// Mitsubishi GX Works2 project: infinite   PLC: Q03UDV

PROGRAM MAIN
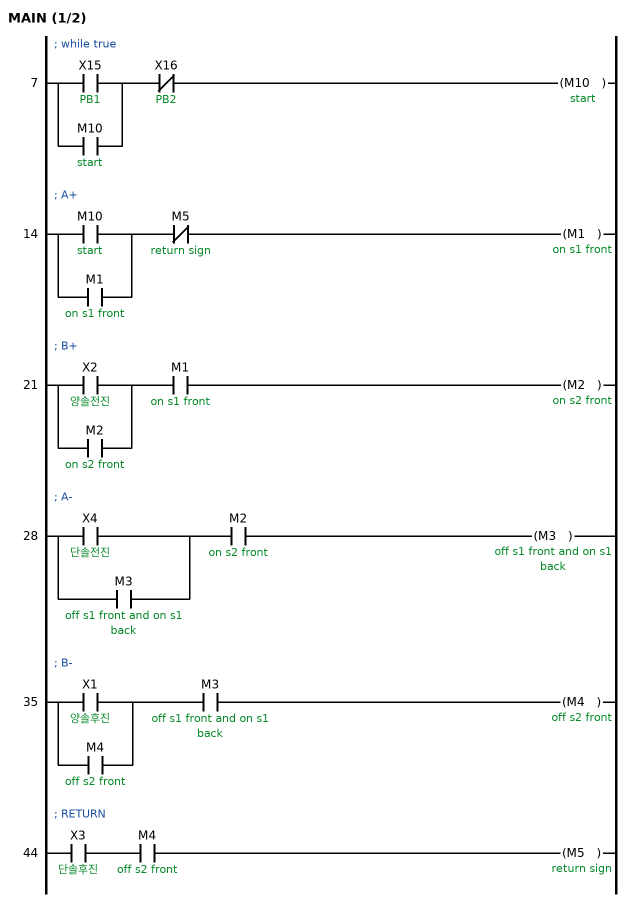
; while true
7     LD      X15  ; PB1
      OR      M10  ; start
      ANI     X16  ; PB2
      OUT     M10  ; start
; A+
14    LD      M10  ; start
      OR      M1  ; on s1 front
      ANI     M5  ; return sign
      OUT     M1  ; on s1 front
; B+
21    LD      X2  ; 양솔전진
      OR      M2  ; on s2 front
      AND     M1  ; on s1 front
      OUT     M2  ; on s2 front
; A-
28    LD      X4  ; 단솔전진
      OR      M3  ; off s1 front and on s1 back
      AND     M2  ; on s2 front
      OUT     M3  ; off s1 front and on s1 back
; B-
35    LD      X1  ; 양솔후진
      OR      M4  ; off s2 front
      AND     M3  ; off s1 front and on s1 back
      OUT     M4  ; off s2 front
; RETURN
44    LD      X3  ; 단솔후진
      AND     M4  ; off s2 front
      OUT     M5  ; return sign
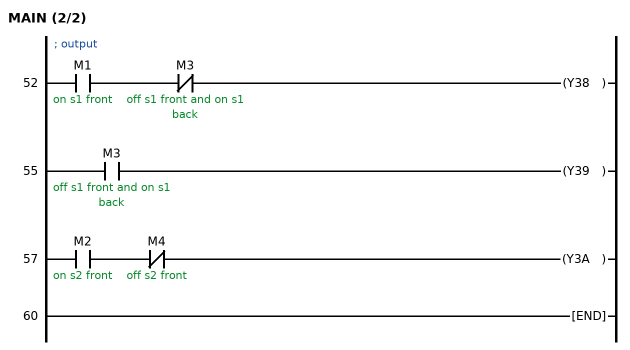
; output
52    LD      M1  ; on s1 front
      ANI     M3  ; off s1 front and on s1 back
      OUT     Y38
55    LD      M3  ; off s1 front and on s1 back
      OUT     Y39
57    LD      M2  ; on s2 front
      ANI     M4  ; off s2 front
      OUT     Y3A
60    END
END_PROGRAM
